    rq_wait_ft_sensor_steady(2000)
    zero_ftsensor()
    sleep(0.1)
    # end: URCap Program Node
    # begin: URCap Program Node
    #   Source: Robotiq_Copilot, 1.22.1.14215, Robotiq Inc.
    #   Type: Find Surface
    $ 103 "Find Surface"
    zero_ftsensor()
    sleep(0.1)
    surface_found = rq_linear_search_urcap("Z+", 10.000, 0.005000, 0.100000, 1)
    storevar.setvariablepose("rq_findSurface_2740b15b-e82c-49d5-a06f-9d0df3e3c4e7_exitPosition", get_actual_tcp_pose())
    $ 104 "'Add Stop conditions from the Find Surface node'" "noBreak"
    # 'Add Stop conditions from the Find Surface node'
    # end: URCap Program Node
    # begin: URCap Program Node
    #   Source: Robotiq_Copilot, 1.22.1.14215, Robotiq Inc.
    #   Type: Finishing Tool Control
    $ 105 "Start tool"
    set_standard_digital_out(0, True)
    # end: URCap Program Node
    $ 106 "Wait: 0.5"
    sleep(0.5)
    $ 107 "Force"
    sleep(0.02)
    zero_ftsensor()
    force_mode(tool_pose(), [0, 0, 1, 0, 0, 0], [0.0, 0.0, 5.0, 0.0, 0.0, 0.0], 2, [0.1, 0.1, 0.15, 0.3490658503988659, 0.3490658503988659, 0.3490658503988659])
    $ 108 "Waypoint_7" "noBreak"
    set_tcp(p[0.00318,0.11464,0.09820000000000001,-0.7853981633974483,0.0,0.0])
    movel(pose_trans(CubeFront, pose_trans(p[.002249871974, -.169402369556, .608081756259, .020435046430, 2.223511403835, 2.209446612627], Waypoint_7_p)), a=1.2, v=0.05)
    end_force_mode()
    stopl(5.0)
    # begin: URCap Program Node
    #   Source: Robotiq_Copilot, 1.22.1.14215, Robotiq Inc.
    #   Type: Finishing Tool Control
    $ 109 "Stop tool"
    set_standard_digital_out(0, False)
    # end: URCap Program Node
    $ 110 "Waypoint_13" "breakAfter"
    set_tcp(p[0.00318,0.11464,0.09820000000000001,-0.7853981633974483,0.0,0.0])
    movel(pose_trans(CubeFront, pose_trans(p[-.002001169423, -.178123008725, .618090231485, -1.568699287997, .013964727372, .007428573496], Waypoint_13_p)), a=1.2, v=0.25)
    $ 111 "Waypoint_9" "breakAfter"
    set_tcp(p[0.00318,0.11464,0.09820000000000001,-0.7853981633974483,0.0,0.0])
    movel(pose_trans(CubeFront, pose_trans(p[-.002001169423, -.178123008725, .618090231485, -1.568699287997, .013964727372, .007428573496], Waypoint_9_p)), a=1.2, v=0.25)
    $ 112 "Clear" "breakAfter"
    set_tcp(p[0.00318,0.11464,0.09820000000000001,-0.7853981633974483,0.0,0.0])
    movel(pose_trans(CubeFront, pose_trans(p[.196772760295, -.286594875311, .585860142249, -1.215980175001, -1.189689100159, -1.189727544600], Clear_p)), a=1.2, v=0.25)
  end
  def SprayFront():
    $ 113 "SprayFront" "noBreak"
    $ 114 "SprayFront"
    $ 115 "MoveJ"
    $ 116 "SprayClear" "breakAfter"
    set_tcp(p[0.020839023181949995,-0.027139950822234082,0.10599373590389219,0.12258870209179472,1.1769383890382668,2.869747076630172])
    movej(get_inverse_kin(pose_trans(SprayPlane, pose_trans(p[.108036142494, -.305202473770, .810091201248, -1.216647948939, 1.210557871618, 1.204123812639], SprayClear_p)), qnear=SprayClear_q), a=1.3962634015954636, v=1.0471975511965976)
    $ 117 "MoveJ"
    $ 118 "Waypoint_10" "breakAfter"
    set_tcp(p[0.020839023181949995,-0.027139950822234082,0.10599373590389219,0.12258870209179472,1.1769383890382668,2.869747076630172])
    movej(get_inverse_kin(pose_trans(SprayPlane, pose_trans(p[.380158499114, -.183027591855, .571104219868, -1.574901506950, .032921162495, .010611987369], Waypoint_10_p)), qnear=Waypoint_10_q), a=1.3962634015954636, v=1.0471975511965976)
    $ 119 "Set DO[4]=On"
    set_standard_digital_out(4, True)
    $ 120 "MoveL"
    $ 121 "Waypoint_12" "breakAfter"
    movel(pose_trans(SprayPlane, pose_trans(p[.380158499114, -.183027591855, .571104219868, -1.574901506950, .032921162495, .010611987369], Waypoint_12_p)), a=1.2, v=0.1)
    $ 122 "Set DO[4]=Off"
    set_standard_digital_out(4, False)
    $ 123 "MoveJ"
    $ 124 "Waypoint_21" "breakAfter"
    set_tcp(p[0.020839023181949995,-0.027139950822234082,0.10599373590389219,0.12258870209179472,1.1769383890382668,2.869747076630172])
    movej(get_inverse_kin(pose_trans(SprayPlane, pose_trans(p[.380158499114, -.183027591855, .571104219868, -1.574901506950, .032921162495, .010611987369], Waypoint_21_p)), qnear=Waypoint_21_q), a=1.3962634015954636, v=1.0471975511965976)
    $ 125 "Set DO[4]=On"
    set_standard_digital_out(4, True)
    $ 126 "MoveL"
    $ 127 "Waypoint_22" "breakAfter"
    set_tcp(p[0.020839023181949995,-0.027139950822234082,0.10599373590389219,0.12258870209179472,1.1769383890382668,2.869747076630172])
    movel(pose_trans(SprayPlane, pose_trans(p[.380158499114, -.183027591855, .571104219868, -1.574901506950, .032921162495, .010611987369], Waypoint_22_p)), a=1.2, v=0.1)
    $ 128 "Set DO[4]=Off"
    set_standard_digital_out(4, False)
    $ 129 "MoveJ"
    $ 130 "Waypoint_23" "breakAfter"
    set_tcp(p[0.020839023181949995,-0.027139950822234082,0.10599373590389219,0.12258870209179472,1.1769383890382668,2.869747076630172])
    movej(get_inverse_kin(pose_trans(SprayPlane, pose_trans(p[.200894234219, -.299948761986, .678711619414, -1.215428189557, 1.212361481441, 1.193485326269], Waypoint_23_p)), qnear=Waypoint_23_q), a=1.3962634015954636, v=1.0471975511965976)
    $ 131 "Set DO[4]=On"
    set_standard_digital_out(4, True)
    $ 132 "MoveL"
    $ 133 "Waypoint_24" "breakAfter"
    set_tcp(p[0.020839023181949995,-0.027139950822234082,0.10599373590389219,0.12258870209179472,1.1769383890382668,2.869747076630172])
    movel(pose_trans(SprayPlane, pose_trans(p[.200894234219, -.299948761986, .678711619414, -1.215428189557, 1.212361481441, 1.193485326269], Waypoint_24_p)), a=1.2, v=0.1)
    $ 134 "Set DO[4]=Off"
    set_standard_digital_out(4, False)
    $ 135 "MoveJ"
    $ 136 "Waypoint_38" "breakAfter"
    set_tcp(p[0.020839023181949995,-0.027139950822234082,0.10599373590389219,0.12258870209179472,1.1769383890382668,2.869747076630172])
    movej(get_inverse_kin(pose_trans(SprayPlane, pose_trans(p[.152076837040, -.186455621862, .570552501782, -1.567181840228, .028822735400, .008142754325], Waypoint_38_p)), qnear=Waypoint_38_q), a=1.3962634015954636, v=1.0471975511965976)
    $ 137 "Set DO[4]=On"
    set_standard_digital_out(4, True)
    $ 138 "MoveL"
    $ 139 "Waypoint_25" "breakAfter"
    set_tcp(p[0.020839023181949995,-0.027139950822234082,0.10599373590389219,0.12258870209179472,1.1769383890382668,2.869747076630172])
    movel(pose_trans(SprayPlane, pose_trans(p[.380158499114, -.183027591855, .571104219868, -1.574901506950, .032921162495, .010611987369], Waypoint_25_p)), a=1.2, v=0.1)
    $ 140 "Set DO[4]=Off"
    set_standard_digital_out(4, False)
    $ 141 "MoveJ"
    $ 142 "SprayClear" "breakAfter"
    set_tcp(p[0.020839023181949995,-0.027139950822234082,0.10599373590389219,0.12258870209179472,1.1769383890382668,2.869747076630172])
    movej(get_inverse_kin(pose_trans(SprayPlane, pose_trans(p[.108036142494, -.305202473770, .810091201248, -1.216647948939, 1.210557871618, 1.204123812639], SprayClear_p)), qnear=SprayClear_q), a=1.3962634015954636, v=1.0471975511965976)
  end
  def SprayRebate():
    $ 143 "SprayRebate" "noBreak"
    $ 144 "SprayRebate"
    $ 145 "MoveJ"
    $ 146 "SprayClear" "breakAfter"
    set_tcp(p[0.020839023181949995,-0.027139950822234082,0.10599373590389219,0.12258870209179472,1.1769383890382668,2.869747076630172])
    movej(get_inverse_kin(pose_trans(SprayPlane, pose_trans(p[.108036142494, -.305202473770, .810091201248, -1.216647948939, 1.210557871618, 1.204123812639], SprayClear_p)), qnear=SprayClear_q), a=1.3962634015954636, v=1.0471975511965976)
    $ 147 "MoveJ"
    $ 148 "Waypoint_28" "breakAfter"
    set_tcp(p[0.020839023181949995,-0.027139950822234082,0.10599373590389219,0.12258870209179472,1.1769383890382668,2.869747076630172])
    movej(get_inverse_kin(pose_trans(SprayPlane, pose_trans(p[-.002001169423, -.178123008725, .618090231485, -1.568699287997, .013964727372, .007428573496], Waypoint_28_p)), qnear=Waypoint_28_q), a=1.3962634015954636, v=1.0471975511965976)
    $ 149 "Set DO[4]=On"
    set_standard_digital_out(4, True)
    $ 150 "MoveL"
    $ 151 "Waypoint_27" "breakAfter"
    set_tcp(p[0.020839023181949995,-0.027139950822234082,0.10599373590389219,0.12258870209179472,1.1769383890382668,2.869747076630172])
    movel(pose_trans(SprayPlane, pose_trans(p[-.002001169423, -.178123008725, .618090231485, -1.568699287997, .013964727372, .007428573496], Waypoint_27_p)), a=1.2, v=0.1)
    $ 152 "Set DO[4]=Off"
    set_standard_digital_out(4, False)
    $ 153 "MoveJ"
    $ 154 "Waypoint_29" "breakAfter"
    set_tcp(p[0.020839023181949995,-0.027139950822234082,0.10599373590389219,0.12258870209179472,1.1769383890382668,2.869747076630172])
    movej(get_inverse_kin(pose_trans(SprayPlane, pose_trans(p[-.002001169423, -.178123008725, .618090231485, -1.568699287997, .013964727372, .007428573496], Waypoint_29_p)), qnear=Waypoint_29_q), a=1.3962634015954636, v=1.0471975511965976)
    $ 155 "Set DO[4]=On"
    set_standard_digital_out(4, True)
    $ 156 "MoveL"
    $ 157 "Waypoint_30" "breakAfter"
    set_tcp(p[0.020839023181949995,-0.027139950822234082,0.10599373590389219,0.12258870209179472,1.1769383890382668,2.869747076630172])
    movel(pose_trans(SprayPlane, pose_trans(p[-.002001169423, -.178123008725, .618090231485, -1.568699287997, .013964727372, .007428573496], Waypoint_30_p)), a=1.2, v=0.1)
    $ 158 "Set DO[4]=Off"
    set_standard_digital_out(4, False)
    $ 159 "MoveJ"
    $ 160 "SprayClear" "breakAfter"
    set_tcp(p[0.020839023181949995,-0.027139950822234082,0.10599373590389219,0.12258870209179472,1.1769383890382668,2.869747076630172])
    movej(get_inverse_kin(pose_trans(SprayPlane, pose_trans(p[.108036142494, -.305202473770, .810091201248, -1.216647948939, 1.210557871618, 1.204123812639], SprayClear_p)), qnear=SprayClear_q), a=1.3962634015954636, v=1.0471975511965976)
    $ 161 "MoveJ"
    $ 162 "Waypoint_32" "breakAfter"
    set_tcp(p[0.020839023181949995,-0.027139950822234082,0.10599373590389219,0.12258870209179472,1.1769383890382668,2.869747076630172])
    movej(get_inverse_kin(pose_trans(SprayPlane, pose_trans(p[-.002001169423, -.178123008725, .618090231485, -1.568699287997, .013964727372, .007428573496], Waypoint_32_p)), qnear=Waypoint_32_q), a=1.3962634015954636, v=1.0471975511965976)
    $ 163 "Set DO[4]=On"
    set_standard_digital_out(4, True)
    $ 164 "MoveL"
    $ 165 "Waypoint_33" "breakAfter"
    set_tcp(p[0.020839023181949995,-0.027139950822234082,0.10599373590389219,0.12258870209179472,1.1769383890382668,2.869747076630172])
    movel(pose_trans(SprayPlane, pose_trans(p[-.002001169423, -.178123008725, .618090231485, -1.568699287997, .013964727372, .007428573496], Waypoint_33_p)), a=1.2, v=0.1)
    $ 166 "Set DO[4]=Off"
    set_standard_digital_out(4, False)
    $ 167 "MoveJ"
    $ 168 "SprayClear" "breakAfter"
    set_tcp(p[0.020839023181949995,-0.027139950822234082,0.10599373590389219,0.12258870209179472,1.1769383890382668,2.869747076630172])
    movej(get_inverse_kin(pose_trans(SprayPlane, pose_trans(p[.108036142494, -.305202473770, .810091201248, -1.216647948939, 1.210557871618, 1.204123812639], SprayClear_p)), qnear=SprayClear_q), a=1.3962634015954636, v=1.0471975511965976)
  end
  def SandFront():
    $ 169 "SandFront" "noBreak"
    $ 170 "sandFront"
    $ 171 "MoveJ"
    $ 172 "Waypoint_35" "breakAfter"
    set_tcp(p[0.00318,0.11464,0.09820000000000001,-0.7853981633974483,0.0,0.0])
    movej(get_inverse_kin(pose_trans(Work, pose_trans(p[.156676362668, -.286472317303, .691031878722, -1.202994956474, -1.209679317392, -1.217118867263], Waypoint_35_p)), qnear=Waypoint_35_q), a=1.3962634015954636, v=1.0471975511965976)
    $ 173 "MoveL"
    $ 174 "Waypoint_1" "breakAfter"
    set_tcp(p[0.00318,0.11464,0.09820000000000001,-0.7853981633974483,0.0,0.0])
    movel(pose_trans(Work, pose_trans(p[-.005597006121, -.192408094989, .653246871754, -1.571622694982, -.002967386491, .002471774867], Waypoint_1_p)), a=1.2, v=0.25)
    # begin: URCap Program Node
    #   Source: Robotiq_Copilot, 1.22.1.14215, Robotiq Inc.
    #   Type: Zero FT Sensor
    $ 175 "Zero FT Sensor"

    rq_wait_ft_sensor_steady(2000)
    zero_ftsensor()
    sleep(0.1)
    # end: URCap Program Node
    # begin: URCap Program Node
    #   Source: Robotiq_Copilot, 1.22.1.14215, Robotiq Inc.
    #   Type: Find Surface
    $ 176 "Find Surface"
    surface_found = rq_linear_search_urcap("Z+", 10.000, 0.005000, 0.100000, 1)
    storevar.setvariablepose("rq_findSurface_ef18b09c-0892-4a94-86ec-4438695763ad_exitPosition", get_actual_tcp_pose())
    $ 177 "'Add Stop conditions from the Find Surface node'" "noBreak"
    # 'Add Stop conditions from the Find Surface node'
    # end: URCap Program Node
    # begin: URCap Program Node
    #   Source: Robotiq_Copilot, 1.22.1.14215, Robotiq Inc.
    #   Type: Finishing Tool Control
    $ 178 "Start tool"
    set_standard_digital_out(0, True)
    # end: URCap Program Node
    $ 179 "Wait: 0.5"
    sleep(0.5)
    $ 180 "MoveL"
    $ 181 "Force"
    sleep(0.02)
    zero_ftsensor()
    force_mode(tool_pose(), [0, 0, 1, 0, 0, 0], [0.0, 0.0, 5.0, 0.0, 0.0, 0.0], 2, [0.1, 0.1, 0.15, 0.3490658503988659, 0.3490658503988659, 0.3490658503988659])
    $ 182 "Waypoint_34" "noBreak"
    set_tcp(p[0.00318,0.11464,0.09820000000000001,-0.7853981633974483,0.0,0.0])
    movel(pose_trans(Work, pose_trans(p[.002249871974, -.169402369556, .608081756259, .020435046430, 2.223511403835, 2.209446612627], Waypoint_34_p)), a=1.2, v=0.06)
    $ 183 "Waypoint_37" "noBreak"
    set_tcp(p[0.00318,0.11464,0.09820000000000001,-0.7853981633974483,0.0,0.0])
    movel(pose_trans(Work, pose_trans(p[.002249871974, -.169402369556, .608081756259, .020435046430, 2.223511403835, 2.209446612627], Waypoint_37_p)), a=1.2, v=0.06)
    $ 184 "Waypoint_36" "noBreak"
    set_tcp(p[0.00318,0.11464,0.09820000000000001,-0.7853981633974483,0.0,0.0])
    movel(pose_trans(Work, pose_trans(p[.002249871974, -.169402369556, .608081756259, .020435046430, 2.223511403835, 2.209446612627], Waypoint_36_p)), a=1.2, v=0.06)
    $ 185 "Waypoint_1" "noBreak"
    set_tcp(p[0.00318,0.11464,0.09820000000000001,-0.7853981633974483,0.0,0.0])
    movel(pose_trans(Work, pose_trans(p[-.005597006121, -.192408094989, .653246871754, -1.571622694982, -.002967386491, .002471774867], Waypoint_1_p)), a=1.2, v=0.06)
    # begin: URCap Program Node
    #   Source: Robotiq_Copilot, 1.22.1.14215, Robotiq Inc.
    #   Type: Finishing Tool Control
    $ 186 "Stop tool" "noBreak"
    set_standard_digital_out(0, False)
    # end: URCap Program Node
    end_force_mode()
    stopl(5.0)
    $ 187 "Direction: Tool Z-"
    global move_thread_flag_187=0
    thread move_thread_187():
      enter_critical
      move_thread_flag_187 = 1
      local towardsPos=calculate_point_to_move_towards(get_forward_kin(), [0.0,0.0,-1.0], 0.025)
      movel(towardsPos, a=1.2, v=0.06)
      move_thread_flag_187 = 2
      exit_critical
    end
    move_thread_flag_187 = 0
    move_thread_han_187 = run move_thread_187()
    while (True):
      sleep(1.0E-10)
      if (move_thread_flag_187 > 1):
        join move_thread_han_187
        $ 188 "Until (distance)"
        break
      end
      sync()
    end
    $ 189 "MoveJ"
    $ 190 "Waypoint_35" "breakAfter"
    movej(get_inverse_kin(pose_trans(Work, pose_trans(p[.156676362668, -.286472317303, .691031878722, -1.202994956474, -1.209679317392, -1.217118867263], Waypoint_35_p)), qnear=Waypoint_35_q), a=1.3962634015954636, v=1.0471975511965976)
  end
  def StartSpray():
    $ 191 "StartSpray" "noBreak"
    $ 192 "Set DO[1]=On"
    set_standard_digital_out(1, True)
    $ 193 "Wait: 0.3"
    sleep(0.3)
  end
  def stopSpray():
    $ 194 "stopSpray" "noBreak"
    $ 195 "Set DO[1]=Off"
    set_standard_digital_out(1, False)
    $ 196 "Wait: 0.3"
    sleep(0.3)
  end
  thread EventThread():
    while (True):
      if (get_standard_digital_in(0) ==   False  ):
        $ 57 "Set DO[0]=Off"
        set_standard_digital_out(0, False)
        $ 58 "Set DO[1]=Off"
        set_standard_digital_out(1, False)
        $ 59 "Halt"
        halt
      elif (get_standard_digital_in(1) ==   True  ):
        $ 61 "readyFrontSand≔ True "
        global readyFrontSand=  True
      elif (get_standard_digital_in(2) ==   True  ):
        $ 63 "readyBackSand≔ True "
        global readyBackSand=  True
        $ 64 "Set DO[5]=On"
        set_standard_digital_out(5, True)
      elif (get_standard_digital_in(3) ==   True  ):
        $ 66 "readySpray≔ True "
        global readySpray=  True
      end
      sync()
    end
  end
  eventThread = run EventThread()
  while (True):
    $ 2 "Robot Program"
    $ 3 "Main"
    $ 4 "If readyFrontSand≟ True "
    global thread_flag_4=0
    thread Thread_if_4():
      $ 5 "MoveJ"
      $ 6 "Clear" "breakAfter"
      set_tcp(p[0.00318,0.11464,0.09820000000000001,-0.7853981633974483,0.0,0.0])
      movej(get_inverse_kin(pose_trans(CubeFront, pose_trans(p[.196772760295, -.286594875311, .585860142249, -1.215980175001, -1.189689100159, -1.189727544600], Clear_p)), qnear=Clear_q), a=1.3962634015954636, v=1.0471975511965976)
      # begin: URCap Program Node
      #   Source: Robotiq_Copilot, 1.22.1.14215, Robotiq Inc.
      #   Type: Zero FT Sensor
      $ 7 "Zero FT Sensor"

      rq_wait_ft_sensor_steady(2000)
      zero_ftsensor()
      sleep(0.1)
      # end: URCap Program Node
      $ 8 "Work≔CubeFront"
      global Work=CubeFront
      $ 9 "Call SandFront"
      SandFront()
      $ 10 "Call SandRebate"
      SandRebate()
      $ 11 "readyFrontSand≔ False "
      global readyFrontSand=  False
      thread_flag_4 = 1
    end
    if (readyFrontSand ==   True  ):
      global thread_handler_4=run Thread_if_4()
      while (thread_flag_4 == 0):
        if not(readyFrontSand ==   True  ):
          kill thread_handler_4
          thread_flag_4 = 2
        else:
          sync()
        end
      end
    else:
      thread_flag_4 = 2
    end
    $ 12 "If readyBackSand≟ True "
    global thread_flag_12=0
    thread Thread_if_12():
      $ 13 "Work≔CubeFront"
      global Work=CubeFront
      $ 14 "Call SandFront"
      SandFront()
      $ 15 "readyBackSand≔ False "
      global readyBackSand=  False
      $ 16 "Set DO[5]=Off"
      set_standard_digital_out(5, False)
      thread_flag_12 = 1
    end
    if (readyBackSand ==   True  ):
      global thread_handler_12=run Thread_if_12()
      while (thread_flag_12 == 0):
        if not(readyBackSand ==   True  ):
          kill thread_handler_12
          thread_flag_12 = 2
        else:
          sync()
        end
      end
    else:
      thread_flag_12 = 2
    end
    $ 17 "If readySpray≟ True "
    global thread_flag_17=0
    thread Thread_if_17():
      $ 18 "MoveJ"
      $ 19 "SprayClear" "breakAfter"
      set_tcp(p[0.020839023181949995,-0.027139950822234082,0.10599373590389219,0.12258870209179472,1.1769383890382668,2.869747076630172])
      movej(get_inverse_kin(pose_trans(SprayPlane, pose_trans(p[.108036142494, -.305202473770, .810091201248, -1.216647948939, 1.210557871618, 1.204123812639], SprayClear_p)), qnear=SprayClear_q), a=1.3962634015954636, v=1.0471975511965976)
      # begin: URCap Program Node
      #   Source: Robotiq_Copilot, 1.22.1.14215, Robotiq Inc.
      #   Type: Zero FT Sensor
      $ 20 "Zero FT Sensor"

      rq_wait_ft_sensor_steady(2000)
      zero_ftsensor()
      sleep(0.1)
      # end: URCap Program Node
      $ 21 "Call SprayFront"
      SprayFront()
      $ 22 "Call SprayRebate"
      SprayRebate()
      $ 23 "readySpray≔ False "
      global readySpray=  False
      thread_flag_17 = 1
    end
    if (readySpray ==   True  ):
      global thread_handler_17=run Thread_if_17()
      while (thread_flag_17 == 0):
        if not(readySpray ==   True  ):
          kill thread_handler_17
          thread_flag_17 = 2
        else:
          sync()
        end
      end
    else:
      thread_flag_17 = 2
    end
  end
end
